// TIA Portal project "通讯练习" (V20)

(* hardware
DEVICE "S7-1200 station_1"  S7-1200 Station
   slot 0: "Rack_0"  S7-1200 Rack  Rack  V1.0
   slot 1: "PLC_left"  CPU 1215C DC/DC/DC  6ES7 215-1AG40-0XB0  V4.6
DEVICE "S7-1200 station_2"  S7-1200 Station
   slot 0: "Rack_0"  S7-1200 Rack  Rack  V1.0
   slot 1: "PLC_right"  CPU 1215C DC/DC/DC  6ES7 215-1AG40-0XB0  V4.6
DEVICE "S7-1200 station_3"  S7-1200 Station
   slot 0: "Rack_0"  S7-1200 Rack  Rack  V1.0
   slot 1: "PLC_middle"  CPU 1215C DC/DC/DC  6ES7 215-1AG40-0XB0  V4.6
*)

// ===== PLC "PLC_left"  CPU 1215C DC/DC/DC =====

VAR_GLOBAL   // PLC tag table "默认变量表"
   "System_Byte" AT %MB1 : Byte;
   "FirstScan" AT %M1.0 : Bool;
   "DiagStatusUpdate" AT %M1.1 : Bool;
   "AlwaysTRUE" AT %M1.2 : Bool;
   "AlwaysFALSE" AT %M1.3 : Bool;
   "Clock_Byte" AT %MB0 : Byte;
   "Clock_10Hz" AT %M0.0 : Bool;
   "Clock_5Hz" AT %M0.1 : Bool;
   "Clock_2.5Hz" AT %M0.2 : Bool;
   "Clock_2Hz" AT %M0.3 : Bool;
   "Clock_1.25Hz" AT %M0.4 : Bool;
   "Clock_1Hz" AT %M0.5 : Bool;
   "Clock_0.625Hz" AT %M0.6 : Bool;
   "Clock_0.5Hz" AT %M0.7 : Bool;
   "Tag_1" AT %M2.0 : Bool;
END_VAR

DATA_BLOCK "块_1_DB"   // DB2
{ S7_Optimized_Access := 'FALSE' }
VERSION : 0.1
// stored: InstanceOfName 块_1
"块_1"
BEGIN
END_DATA_BLOCK

// folder: System blocks/Program resources

DATA_BLOCK "PLC_left_Send_DB"   // DB1
{ S7_Optimized_Access := 'TRUE' }
VERSION : 0.1
// stored: InstanceOfName TCON_Configured
"TCON_Configured"
BEGIN
   ID := 257;
   ConnectionType := 254;
END_DATA_BLOCK

DATA_BLOCK "PLC_left_Send_DB_1"   // DB3
{ S7_Optimized_Access := 'TRUE' }
AUTHOR : SIMATIC
FAMILY : MC7Plus
NAME : TC_IP_v4
VERSION : 1.0
// stored: InstanceOfName TCON_IP_v4
"TCON_IP_v4"
BEGIN
   ID := 1;
   InterfaceId := 64;
   ActiveEstablished := true;
   LocalPort := 2000;
   RemotePort := 2011;
   RemoteAddress.ADDR[1] := 192;
   RemoteAddress.ADDR[2] := 168;
   RemoteAddress.ADDR[4] := 11;
END_DATA_BLOCK

// folder: (top level)

FUNCTION_BLOCK "块_1"   // FB1, LAD
{ S7_Optimized_Access := 'FALSE' }
VERSION : 0.1
   VAR
      MB_CLIENT_Instance : MB_CLIENT;
      modbus_tcp_config : TCON_IP_v4;
      写入的数据 : Array[0..10] of DInt;
      读取的数据 : Array[0..10] of DInt;
      modbus_tcp_config_r : TCON_IP_v4;
      MB_CLIENT_Instance_1 : MB_CLIENT;
      TSEND_C_Instance : TSEND_C;
   END_VAR
   VAR_TEMP   // added for the SCL form of the ladder/FBD networks
      _w1 : Bool;
   END_VAR
   // modbus_tcp_config.ActiveEstablished := 1;
   // modbus_tcp_config.RemoteAddress.ADDR[1] := 192;
   // modbus_tcp_config.RemoteAddress.ADDR[2] := 168;
   // modbus_tcp_config.RemoteAddress.ADDR[3] := 0;
   // modbus_tcp_config.RemoteAddress.ADDR[4] := 11;
   // modbus_tcp_config.RemotePort := 2011;
   // modbus_tcp_config.LocalPort := 2000;
   // modbus_tcp_config_r.InterfaceId := 64;
   // modbus_tcp_config_r.ID := 4;
   // modbus_tcp_config_r.RemoteAddress.ADDR[1] := 192;
   // modbus_tcp_config_r.RemoteAddress.ADDR[2] := 168;
   // modbus_tcp_config_r.RemoteAddress.ADDR[3] := 0;
   // modbus_tcp_config_r.RemoteAddress.ADDR[4] := 21;
   // modbus_tcp_config_r.RemotePort := 2022;
   // modbus_tcp_config_r.LocalPort := 2001;
   // modbus_tcp_config_r.ActiveEstablished := 1;
   // modbus_tcp_config.InterfaceId := 64;
   // modbus_tcp_config.ID := 6;
BEGIN

REGION Network 1
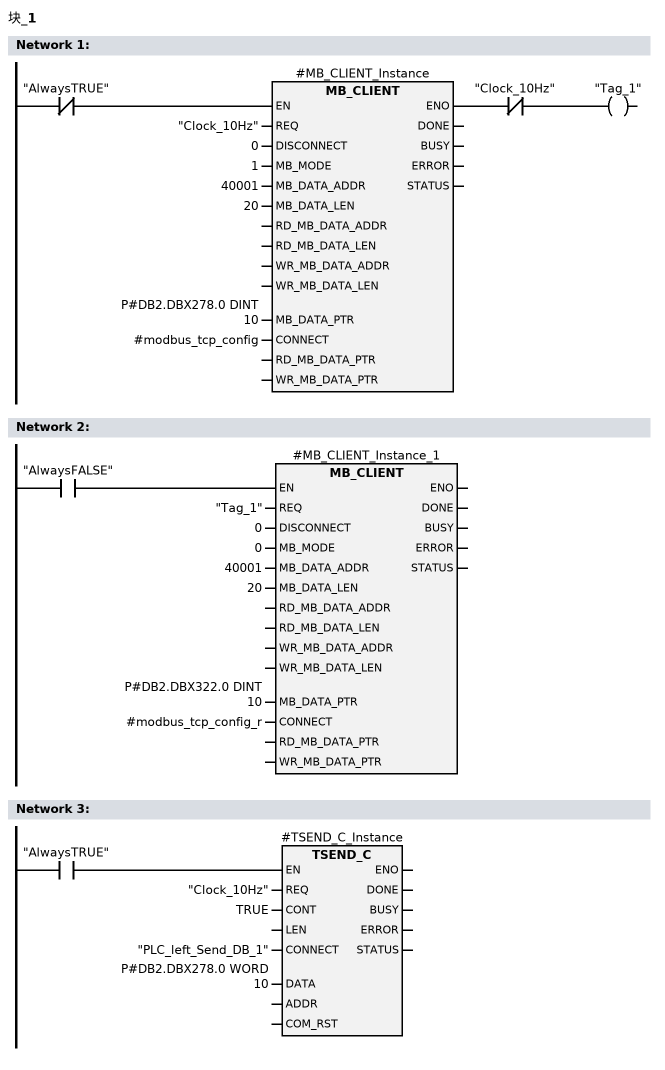
   // ENO of a box is taken as its EN; it also drops when the box reports an error
   #_w1 := NOT "AlwaysTRUE";
   IF #_w1 THEN
       #MB_CLIENT_Instance(REQ := "Clock_10Hz",   // MB_CLIENT
                           DISCONNECT := 0,
                           MB_MODE := 1,
                           MB_DATA_ADDR := 40001,
                           MB_DATA_LEN := 20,
                           MB_DATA_PTR := P#DB2.DBX278.0 DINT 10,
                           CONNECT := #modbus_tcp_config);
   END_IF;
   "Tag_1" := #_w1 AND NOT "Clock_10Hz";
END_REGION

REGION Network 2
   IF "AlwaysFALSE" THEN
       #MB_CLIENT_Instance_1(REQ := "Tag_1",   // MB_CLIENT
                             DISCONNECT := 0,
                             MB_MODE := 0,
                             MB_DATA_ADDR := 40001,
                             MB_DATA_LEN := 20,
                             MB_DATA_PTR := P#DB2.DBX322.0 DINT 10,
                             CONNECT := #modbus_tcp_config_r);
   END_IF;
END_REGION

REGION Network 3
   IF "AlwaysTRUE" THEN
       #TSEND_C_Instance(REQ := "Clock_10Hz",   // TSEND_C
                         CONT := TRUE,
                         CONNECT := "PLC_left_Send_DB_1",
                         DATA := P#DB2.DBX278.0 WORD 10);
   END_IF;
END_REGION
END_FUNCTION_BLOCK

ORGANIZATION_BLOCK "Main"   // OB1, LAD, ProgramCycle
TITLE = "Main Program Sweep (Cycle)"
{ S7_Optimized_Access := 'TRUE' }
VERSION : 0.1
   VAR_INPUT
      Initial_Call : Bool;   // Initial call of this OB
      Remanence : Bool;   // =True, if remanent data are available
   END_VAR
BEGIN

REGION Network 1
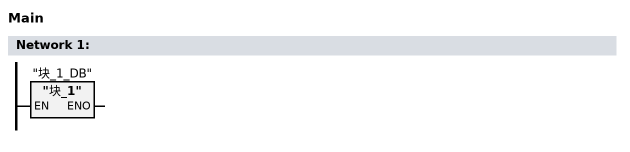
   RUNG wire#powerrail
      "块_1_DB"()
   END_RUNG
   // the same network as SCL:
   "块_1_DB"();   // "块_1"
END_REGION
END_ORGANIZATION_BLOCK

// ===== PLC "PLC_right"  CPU 1215C DC/DC/DC =====

VAR_GLOBAL   // PLC tag table "默认变量表"
   "System_Byte" AT %MB1 : Byte;
   "FirstScan" AT %M1.0 : Bool;
   "DiagStatusUpdate" AT %M1.1 : Bool;
   "AlwaysTRUE" AT %M1.2 : Bool;
   "AlwaysFALSE" AT %M1.3 : Bool;
   "Clock_Byte" AT %MB0 : Byte;
   "Clock_10Hz" AT %M0.0 : Bool;
   "Clock_5Hz" AT %M0.1 : Bool;
   "Clock_2.5Hz" AT %M0.2 : Bool;
   "Clock_2Hz" AT %M0.3 : Bool;
   "Clock_1.25Hz" AT %M0.4 : Bool;
   "Clock_1Hz" AT %M0.5 : Bool;
   "Clock_0.625Hz" AT %M0.6 : Bool;
   "Clock_0.5Hz" AT %M0.7 : Bool;
END_VAR

DATA_BLOCK "块_1_DB"   // DB2
{ S7_Optimized_Access := 'FALSE' }
VERSION : 0.1
// stored: InstanceOfName 块_1
"块_1"
BEGIN
END_DATA_BLOCK

FUNCTION_BLOCK "块_1"   // FB1, LAD
{ S7_Optimized_Access := 'FALSE' }
VERSION : 0.1
   VAR
      modbus_tcp_config_fwm : TCON_IP_v4;
      modbus_tcp_config_frl : TCON_IP_v4;
      MB_SERVER_Instance : MB_SERVER;
      被写入数据 : Array[0..10] of DInt;
      被读取数据 : Array[0..10] of DInt;
      MB_SERVER_Instance_1 : MB_SERVER;
   END_VAR
   // modbus_tcp_config_fwm.ActiveEstablished := 0;
   // modbus_tcp_config_fwm.RemoteAddress.ADDR[1] := 0;
   // modbus_tcp_config_fwm.RemoteAddress.ADDR[2] := 0;
   // modbus_tcp_config_fwm.RemoteAddress.ADDR[3] := 0;
   // modbus_tcp_config_fwm.RemoteAddress.ADDR[4] := 0;
   // modbus_tcp_config_fwm.RemotePort := 2012;
   // modbus_tcp_config_fwm.LocalPort := 2021;
   // modbus_tcp_config_frl.InterfaceId := 64;
   // modbus_tcp_config_frl.ID := 5;
   // modbus_tcp_config_frl.RemotePort := 2001;
   // modbus_tcp_config_frl.LocalPort := 2022;
   // modbus_tcp_config_fwm.InterfaceId := 64;
   // modbus_tcp_config_fwm.ID := 3;
BEGIN

REGION Network 1
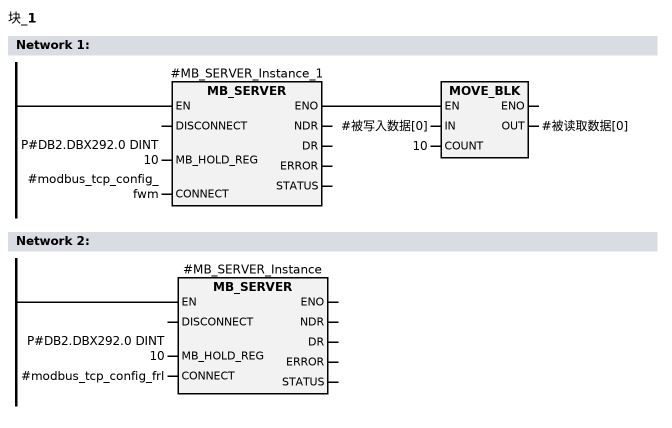
   // ENO of a box is taken as its EN; it also drops when the box reports an error
   #MB_SERVER_Instance_1(MB_HOLD_REG := P#DB2.DBX292.0 DINT 10, CONNECT := #modbus_tcp_config_fwm);   // MB_SERVER
   MOVE_BLK(IN := #被写入数据[0], COUNT := 10, OUT => #被读取数据[0]);
END_REGION

REGION Network 2
   #MB_SERVER_Instance(MB_HOLD_REG := P#DB2.DBX292.0 DINT 10, CONNECT := #modbus_tcp_config_frl);   // MB_SERVER
END_REGION
END_FUNCTION_BLOCK

ORGANIZATION_BLOCK "Main"   // OB1, LAD, ProgramCycle
TITLE = "Main Program Sweep (Cycle)"
{ S7_Optimized_Access := 'TRUE' }
VERSION : 0.1
   VAR_INPUT
      Initial_Call : Bool;   // Initial call of this OB
      Remanence : Bool;   // =True, if remanent data are available
   END_VAR
BEGIN

REGION Network 1
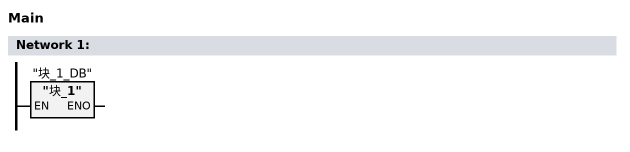
   RUNG wire#powerrail
      "块_1_DB"()
   END_RUNG
   // the same network as SCL:
   "块_1_DB"();   // "块_1"
END_REGION
END_ORGANIZATION_BLOCK

// ===== PLC "PLC_middle"  CPU 1215C DC/DC/DC =====

VAR_GLOBAL   // PLC tag table "默认变量表"
   "System_Byte" AT %MB1 : Byte;
   "FirstScan" AT %M1.0 : Bool;
   "DiagStatusUpdate" AT %M1.1 : Bool;
   "AlwaysTRUE" AT %M1.2 : Bool;
   "AlwaysFALSE" AT %M1.3 : Bool;
   "Clock_Byte" AT %MB0 : Byte;
   "Clock_10Hz" AT %M0.0 : Bool;
   "Clock_5Hz" AT %M0.1 : Bool;
   "Clock_2.5Hz" AT %M0.2 : Bool;
   "Clock_2Hz" AT %M0.3 : Bool;
   "Clock_1.25Hz" AT %M0.4 : Bool;
   "Clock_1Hz" AT %M0.5 : Bool;
   "Clock_0.625Hz" AT %M0.6 : Bool;
   "Clock_0.5Hz" AT %M0.7 : Bool;
END_VAR

DATA_BLOCK "块_1_DB"   // DB2
{ S7_Optimized_Access := 'FALSE' }
VERSION : 0.1
// stored: InstanceOfName 块_1
"块_1"
BEGIN
END_DATA_BLOCK

// folder: System blocks/Program resources

DATA_BLOCK "PLC_middle_Receive_DB"   // DB1
{ S7_Optimized_Access := 'TRUE' }
VERSION : 0.1
// stored: InstanceOfName TCON_Configured
"TCON_Configured"
BEGIN
   ID := 256;
   ConnectionType := 254;
END_DATA_BLOCK

DATA_BLOCK "PLC_middle_Receive_DB_1"   // DB3
{ S7_Optimized_Access := 'TRUE' }
AUTHOR : SIMATIC
FAMILY : MC7Plus
NAME : TC_IP_v4
VERSION : 1.0
// stored: InstanceOfName TCON_IP_v4
"TCON_IP_v4"
BEGIN
   ID := 1;
   InterfaceId := 64;
   LocalPort := 2011;
   RemotePort := 2000;
END_DATA_BLOCK

// folder: (top level)

FUNCTION_BLOCK "块_1"   // FB1, LAD
{ S7_Optimized_Access := 'FALSE' }
VERSION : 0.1
   VAR
      MB_CLIENT_Instance : MB_CLIENT;
      modbus_tcp_config_w : TCON_IP_v4;
      modbus_tcp_config_fw : TCON_IP_v4;
      MB_SERVER_Instance : MB_SERVER;
      被写入数据 : Array[0..10] of DInt;
      写入数据 : Array[0..10] of DInt;
      TRCV_C_Instance : TRCV_C;
   END_VAR
   // modbus_tcp_config_w.ActiveEstablished := 1;
   // modbus_tcp_config_w.RemoteAddress.ADDR[1] := 192;
   // modbus_tcp_config_w.RemoteAddress.ADDR[2] := 168;
   // modbus_tcp_config_w.RemoteAddress.ADDR[3] := 0;
   // modbus_tcp_config_w.RemoteAddress.ADDR[4] := 21;
   // modbus_tcp_config_w.RemotePort := 2021;
   // modbus_tcp_config_w.LocalPort := 2012;
   // modbus_tcp_config_fw.InterfaceId := 64;
   // modbus_tcp_config_fw.ID := 1;
   // modbus_tcp_config_fw.RemotePort := 2000;
   // modbus_tcp_config_fw.LocalPort := 2011;
   // modbus_tcp_config_w.InterfaceId := 64;
   // modbus_tcp_config_w.ID := 2;
BEGIN

REGION Network 1
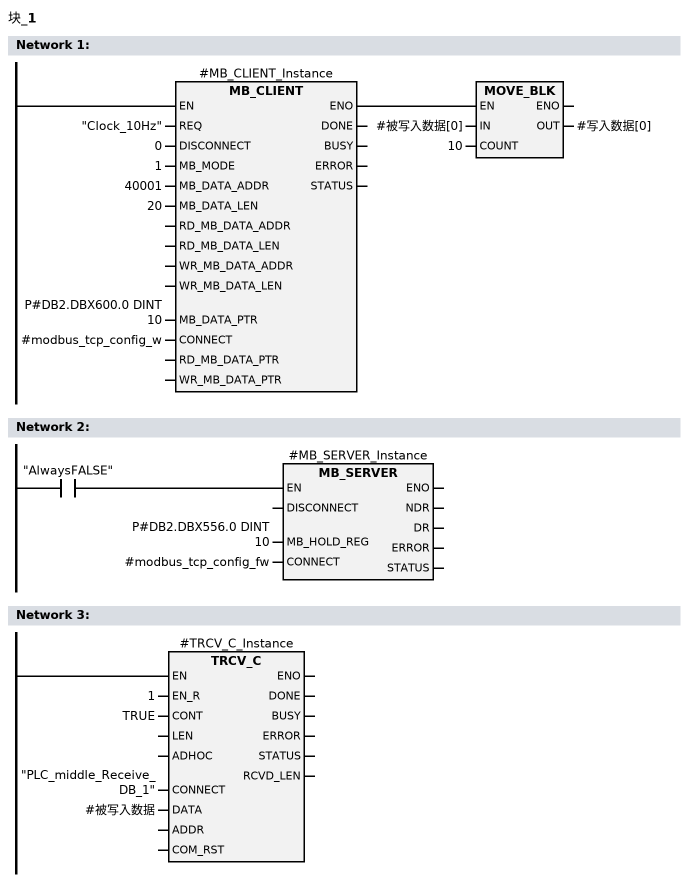
   // ENO of a box is taken as its EN; it also drops when the box reports an error
   #MB_CLIENT_Instance(REQ := "Clock_10Hz",   // MB_CLIENT
                       DISCONNECT := 0,
                       MB_MODE := 1,
                       MB_DATA_ADDR := 40001,
                       MB_DATA_LEN := 20,
                       MB_DATA_PTR := P#DB2.DBX600.0 DINT 10,
                       CONNECT := #modbus_tcp_config_w);
   MOVE_BLK(IN := #被写入数据[0], COUNT := 10, OUT => #写入数据[0]);
END_REGION

REGION Network 2
   IF "AlwaysFALSE" THEN
       #MB_SERVER_Instance(MB_HOLD_REG := P#DB2.DBX556.0 DINT 10, CONNECT := #modbus_tcp_config_fw);   // MB_SERVER
   END_IF;
END_REGION

REGION Network 3
   #TRCV_C_Instance(EN_R := 1, CONT := TRUE, CONNECT := "PLC_middle_Receive_DB_1", DATA := #被写入数据);   // TRCV_C
END_REGION
END_FUNCTION_BLOCK

ORGANIZATION_BLOCK "Main"   // OB1, LAD, ProgramCycle
TITLE = "Main Program Sweep (Cycle)"
{ S7_Optimized_Access := 'TRUE' }
VERSION : 0.1
   VAR_INPUT
      Initial_Call : Bool;   // Initial call of this OB
      Remanence : Bool;   // =True, if remanent data are available
   END_VAR
BEGIN

REGION Network 1
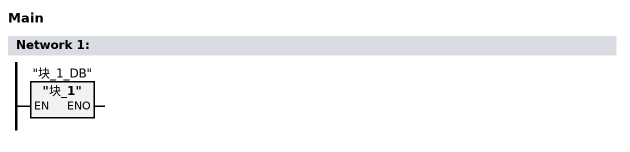
   RUNG wire#powerrail
      "块_1_DB"()
   END_RUNG
   // the same network as SCL:
   "块_1_DB"();   // "块_1"
END_REGION
END_ORGANIZATION_BLOCK